INTERFACE Subject_Interface

METHOD Get_Method : INT
END_METHOD

METHOD Set_Method
VAR_INPUT
	///Value to be set passed as an argument
	num: INT;
END_VAR
END_METHOD

END_INTERFACE

(* stored: Version 1.1.0.1, ProductVersion 3.1.4024.12
   Itf Subject_Interface: Id {9b176648-f559-43a2-83ce-c145c4e85927}
   Method Get_Method: Id {43ef36d3-139e-4bf2-9c1f-5b8936d55187}
   Method Set_Method: Id {3c1b6c87-b1d5-4e04-802e-e3fea42eb71f} *)
